// TIA Portal V16 export
// export: Created 2023-11-14T19:43:19.8365651Z, ExportSetting WithDefaults, DisplayName Totally Integrated Automation Portal, DisplayVersion V16, DisplayName TIA Portal Version Control Interface, DisplayVersion V16, DisplayName TIA Portal Openness, DisplayVersion V16, DisplayName SINAMICS Startdrive Advanced, DisplayVersion V16, DisplayName SINAMICS Startdrive G130, G150, S120, S150, SINAMICS MV, S210, DisplayVersion V16, DisplayName SINAMICS Startdrive G110M, G120, G120C, G120D, G120P, DisplayVersion V16, DisplayName STEP 7 Professional, DisplayVersion V16, DisplayName STEP 7 Safety, DisplayVersion V16, DisplayName WinCC Professional, DisplayVersion V16
VAR_GLOBAL   // PLC tag table "Default tag table"
   Iniciar_Manual AT %I0.0 : Bool;
   Detener_Manual AT %I0.1 : Bool;
   Raw_Temperatura AT %IW64 : Int;
   Raw_Humedad AT %IW66 : Int;
   Deshidratador AT %Q0.0 : Bool;
   Actuador AT %Q0.1 : Bool;
   Ventilador AT %Q0.2 : Bool;
   Resistencias AT %Q0.3 : Bool;
   Sensor_Modbus AT %Q0.4 : Bool;
   Sensor_HT AT %Q0.5 : Bool;
   System_Byte AT %MB1 : Byte;
   FirstScan AT %M1.0 : Bool;
   DiagStatusUpdate AT %M1.1 : Bool;
   AlwaysTRUE AT %M1.2 : Bool;
   AlwaysFALSE AT %M1.3 : Bool;
   Clock_Byte AT %MB0 : Byte;
   Clock_10Hz AT %M0.0 : Bool;
   Clock_5Hz AT %M0.1 : Bool;
   "Clock_2.5Hz" AT %M0.2 : Bool;
   Clock_2Hz AT %M0.3 : Bool;
   "Clock_1.25Hz" AT %M0.4 : Bool;
   Clock_1Hz AT %M0.5 : Bool;
   "Clock_0.625Hz" AT %M0.6 : Bool;
   "Clock_0.5Hz" AT %M0.7 : Bool;
   Control_Byte AT %MB2 : Byte;
   Detener AT %M2.0 : Bool;
   Iniciar AT %M2.1 : Bool;
   Pausar AT %M2.2 : Bool;
   Activar_Deshidratador AT %M2.3 : Bool;
   Limite_Matte AT %M2.6 : Bool;
   Sensor_Modbus_Manual AT %M2.4 : Bool;
   Set_Point_Deshidratador AT %MD4 : Real;
   Set_Point_Humedad AT %MD8 : Real;
   Iniciar_Pulse AT %M40.0 : Bool;
   Detener_Pulse AT %M40.1 : Bool;
   Guardar_Datos AT %M40.2 : Bool;
   Data_Log_Write_Error AT %M40.3 : Bool;
   Data_Log_Write_Busy AT %M40.4 : Bool;
   Data_Log_Write_Done AT %M40.5 : Bool;
   Data_Log_Write_Status AT %MW96 : Word;
   "Clock_0.016Hz" AT %M40.6 : Bool;
   Ret_Val AT %MW98 : Int;
   Sensor_HT_Manual AT %M2.5 : Bool;
   Actuador_Manual AT %M2.7 : Bool;
   Activar_Actuador AT %M3.0 : Bool;
   Tag_1 AT %M41.1 : Bool;
   Habilitar_Matte AT %M3.1 : Bool;
   Set_Point_Limite AT %MD12 : Real;
   Humedad_Material_D11 AT %MD100 : Real;
   Humedad_Material_D13 AT %MD104 : Real;
   Humedad_Material_D16 AT %MD108 : Real;
   Temp_D13 AT %MD114 : Real;
   Temp_Matte AT %MD118 : Real;
   Hum_Matte AT %MD62 : Real;
   Temp_D11 AT %MD112 : Real;
   Temp_Matte_Aux AT %MD66 : Real;
   Clock_Matte_Manual AT %M41.2 : Bool;
   Humedad_Material_D11_Ajuste AT %MD70 : Real;
   Humedad_Material_D13_Ajuste AT %MD74 : Real;
   Humedad_Material_D16_Ajuste AT %MD78 : Real;
   Hum_Matte_Aux AT %MD82 : Real;
   Random_Real_Seconds AT %MD86 : Real;
   Random_Status AT %MW90 : Int;
   Random_Sub_Status AT %MW92 : Int;
   Random_Error AT %M3.2 : Bool;
   Clock_Pulse AT %M3.3 : Bool;
   Randon_Dint_Seconds AT %MD94 : DInt;
   Tiempo_Histeresis_D1 AT %MD14 : Time;
   Set_Point_Deshidratador1_Inicial AT %MD18 : Real;
   Set_Point_Deshidratador1_Intermedia AT %MD22 : Real;
   Set_Point_Deshidratador1_Final AT %MD24 : Real;
   Set_Point_Humedad_D1_Inicial AT %MD28 : Real;
   Set_Point_Humedad_D1_Intermedia AT %MD32 : Real;
   Set_Point_Humedad_D1_Final AT %MD36 : Real;
   Detener_Desde_Modo_Preset AT %M41.3 : Bool;
END_VAR
VAR_GLOBAL CONSTANT   // user constants
   Set_Point_Temp_Default : Real := 55.0;
   Set_Pont_Hum_Default : Real := 5.0;
   Set_Point_Lim_Default : Real := -16.0;
   Aux_Hum_D1 : Real := 10.0;
   Aux_Hum_D4 : Real := 25.0;
   Aux_Hum_D8 : Real := 25.0;
END_VAR
